Yaskawa INFORM job: IO.JBI

/JOB
//NAME IO
//POS
///NPOS 0,0,0,0,0,0
//INST
///DATE 2018/09/12 13:03
///ATTR SC,RW
///GROUP1 RB1,BS1
NOP
DOUT OG#(4) 0
END
